(* IEC 61131-3 sources: eCockpitGit/test_project/src/%F%00 Library/%F%Common Functions/%F%Y AXB/%F%Direct, 9 files *)

(* ---- %POU%FU_lrABFromCordDir.st ---- *)
//This function calculates an a and a b value for a line equation based on given coordinates
// +-----------+----------+----------+-----------------------------------------------------------------------------------------------------------------------+
// |**Version**|**Author**| **Date** |**Changes**                                                                                                            |
// +-----------+----------+----------+-----------------------------------------------------------------------------------------------------------------------+
// | 1         | NSN      | 29-01-19 | Creation                                                                                                              |
// +-----------+----------+----------+-----------------------------------------------------------------------------------------------------------------------+
FUNCTION FU_lrABFromCordDir : BOOL
VAR_IN_OUT
	rX1		:LREAL;
	rX2		:LREAL;
	rY1		:LREAL;
	rY2		:LREAL;
	rA		:LREAL;
	rB		:LREAL;
END_VAR
(*%!%__DELIMITER__%!%*)
//a value is calculated
IF rX2 - rX1 = 0 THEN rA := 0; ELSE rA := (rY2 - rY1) / (rX2 - rX1); END_IF
//b value is calculated
rB			:=		rY1 - (rA * rX1);

(* ---- %POU%FU_lrABXToYDir.st ---- *)
//This function, calculates the y value in a y = a * x + b equation
// +-----------+----------+----------+-----------------------------------------------------------------------------------------------------------------------+
// |**Version**|**Author**| **Date** |**Changes**                                                                                                            |
// +-----------+----------+----------+-----------------------------------------------------------------------------------------------------------------------+
// | 1         | NSN      | 25-07-18 | Creation                                                                                                              |
// +-----------+----------+----------+-----------------------------------------------------------------------------------------------------------------------+
// | 1.1       | NSN      | 29-01-19 | Updated to new format                                                                                                 |
// +-----------+----------+----------+-----------------------------------------------------------------------------------------------------------------------+
FUNCTION FU_lrABXToYDir : BOOL
VAR_IN_OUT
	rX		:LREAL;
	rA		:LREAL;
	rB		:LREAL;
	rY		:LREAL;
END_VAR
(*%!%__DELIMITER__%!%*)
rY	:=		rA * rX + rB;

(* ---- %POU%FU_lrABYToXDir.st ---- *)
//This function, calculates the x value in a x = (y - b) / a equation
// +-----------+----------+----------+-----------------------------------------------------------------------------------------------------------------------+
// |**Version**|**Author**| **Date** |**Changes**                                                                                                            |
// +-----------+----------+----------+-----------------------------------------------------------------------------------------------------------------------+
// | 1         | NSN      | 25-07-18 | Creation                                                                                                              |
// +-----------+----------+----------+-----------------------------------------------------------------------------------------------------------------------+
// | 1.1       | NSN      | 29-01-19 | Updated to new format                                                                                                 |
// +-----------+----------+----------+-----------------------------------------------------------------------------------------------------------------------+
FUNCTION FU_lrABYToXDir : BOOL
VAR_IN_OUT
	rY		:LREAL;
	rA		:LREAL;
	rB		:LREAL;
	rX		:LREAL;
END_VAR
(*%!%__DELIMITER__%!%*)
IF rA <> 0 THEN
	rX	:=		(rY - rB) / rA;
ELSE
	rX	:=		0;
END_IF

(* ---- %POU%FU_rABFromCordDir.st ---- *)
//This function calculates an a and a b value for a line equation based on given coordinates
// +-----------+----------+----------+-----------------------------------------------------------------------------------------------------------------------+
// |**Version**|**Author**| **Date** |**Changes**                                                                                                            |
// +-----------+----------+----------+-----------------------------------------------------------------------------------------------------------------------+
// | 1         | NSN      | 25-07-18 | Creation                                                                                                              |
// +-----------+----------+----------+-----------------------------------------------------------------------------------------------------------------------+
// | 1.1       | NSN      | 29-01-19 | Updated to new format                                                                                                 |
// +-----------+----------+----------+-----------------------------------------------------------------------------------------------------------------------+
FUNCTION FU_rABFromCordDir : BOOL
VAR_IN_OUT
	rX1		:REAL;
	rX2		:REAL;
	rY1		:REAL;
	rY2		:REAL;
	rA		:REAL;
	rB		:REAL;
END_VAR
(*%!%__DELIMITER__%!%*)
//a value is calculated
IF rX2 - rX1 = 0 THEN rA := 0; ELSE rA := (rY2 - rY1) / (rX2 - rX1); END_IF
//b value is calculated
rB			:=		rY1 - (rA * rX1);

(* ---- %POU%FU_rABFromCordDPDir.st ---- *)
//This function calculates an a and a b value for a line equation based on given coordinates
//This is the double precision version, which means all values are converted to LREAL before mathematics
// +-----------+----------+----------+-----------------------------------------------------------------------------------------------------------------------+
// |**Version**|**Author**| **Date** |**Changes**                                                                                                            |
// +-----------+----------+----------+-----------------------------------------------------------------------------------------------------------------------+
// | 1         | NSN      | 29-01-19 | Creation                                                                                                              |
// +-----------+----------+----------+-----------------------------------------------------------------------------------------------------------------------+
FUNCTION FU_rABFromCordDPDir : BOOL
VAR_IN_OUT
	rX1		:REAL;
	rX2		:REAL;
	rY1		:REAL;
	rY2		:REAL;
	rA		:REAL;
	rB		:REAL;
END_VAR
(*%!%__DELIMITER__%!%*)
//a value is calculated
IF TO_LREAL(rX2) - TO_LREAL(rX1) = 0 THEN rA := 0; ELSE rA := TO_REAL((TO_LREAL(rY2) - TO_LREAL(rY1)) / (TO_LREAL(rX2) - TO_LREAL(rX1))); END_IF
//b value is calculated
rB			:=		TO_REAL(TO_LREAL(rY1) - (TO_LREAL(rA) * TO_LREAL(rX1)));

(* ---- %POU%FU_rABXToYDir.st ---- *)
//This function, calculates the y value in a y = a * x + b equation
// +-----------+----------+----------+-----------------------------------------------------------------------------------------------------------------------+
// |**Version**|**Author**| **Date** |**Changes**                                                                                                            |
// +-----------+----------+----------+-----------------------------------------------------------------------------------------------------------------------+
// | 1         | NSN      | 25-07-18 | Creation                                                                                                              |
// +-----------+----------+----------+-----------------------------------------------------------------------------------------------------------------------+
// | 1.1       | NSN      | 29-01-19 | Updated to new format                                                                                                 |
// +-----------+----------+----------+-----------------------------------------------------------------------------------------------------------------------+
FUNCTION FU_rABXToYDir : BOOL
VAR_IN_OUT
	rX		:REAL;
	rA		:REAL;
	rB		:REAL;
	rY		:REAL;
END_VAR
(*%!%__DELIMITER__%!%*)
rY	:=		rA * rX + rB;

(* ---- %POU%FU_rABXToYDPDir.st ---- *)
//This function, calculates the y value in a y = a * x + b equation
//This is the double precision version, which means all values are converted to LREAL before mathematics
// +-----------+----------+----------+-----------------------------------------------------------------------------------------------------------------------+
// |**Version**|**Author**| **Date** |**Changes**                                                                                                            |
// +-----------+----------+----------+-----------------------------------------------------------------------------------------------------------------------+
// | 1         | NSN      | 29-01-19 | Creation                                                                                                              |
// +-----------+----------+----------+-----------------------------------------------------------------------------------------------------------------------+
FUNCTION FU_rABXToYDPDir : BOOL
VAR_IN_OUT
	rX		:REAL;
	rA		:REAL;
	rB		:REAL;
	rY		:REAL;
END_VAR
(*%!%__DELIMITER__%!%*)
rY		:=		TO_REAL(TO_LREAL(rA) * TO_LREAL(rX) + TO_LREAL(rB));

(* ---- %POU%FU_rABYToXDir.st ---- *)
//This function, calculates the x value in a x = (y - b) / a equation
// +-----------+----------+----------+-----------------------------------------------------------------------------------------------------------------------+
// |**Version**|**Author**| **Date** |**Changes**                                                                                                            |
// +-----------+----------+----------+-----------------------------------------------------------------------------------------------------------------------+
// | 1         | NSN      | 25-07-18 | Creation                                                                                                              |
// +-----------+----------+----------+-----------------------------------------------------------------------------------------------------------------------+
// | 1.1       | NSN      | 29-01-19 | Updated to new format                                                                                                 |
// +-----------+----------+----------+-----------------------------------------------------------------------------------------------------------------------+
FUNCTION FU_rABYToXDir : BOOL
VAR_IN_OUT
	rY		:REAL;
	rA		:REAL;
	rB		:REAL;
	rX		:REAL;
END_VAR
(*%!%__DELIMITER__%!%*)
IF rA <> 0 THEN
	rX	:=		(rY - rB) / rA;
ELSE
	rX	:=		0;
END_IF

(* ---- %POU%FU_rABYToXDPDir.st ---- *)
//This function, calculates the x value in a x = (y - b) / a equation
//This is the double precision version, which means all values are converted to LREAL before mathematics
// +-----------+----------+----------+-----------------------------------------------------------------------------------------------------------------------+
// |**Version**|**Author**| **Date** |**Changes**                                                                                                            |
// +-----------+----------+----------+-----------------------------------------------------------------------------------------------------------------------+
// | 1         | NSN      | 29-01-19 | Creation                                                                                                              |
// +-----------+----------+----------+-----------------------------------------------------------------------------------------------------------------------+
FUNCTION FU_rABYToXDPDir : BOOL
VAR_IN_OUT
	rY		:REAL;
	rA		:REAL;
	rB		:REAL;
	rX		:REAL;
END_VAR
(*%!%__DELIMITER__%!%*)
IF rA <> 0 THEN
	rX	:=		TO_REAL((TO_LREAL(rY) - TO_LREAL(rB)) / TO_LREAL(rA));
ELSE
	rX	:=		0;
END_IF
